Universal Robots PolyScope program: PaintTop.urp

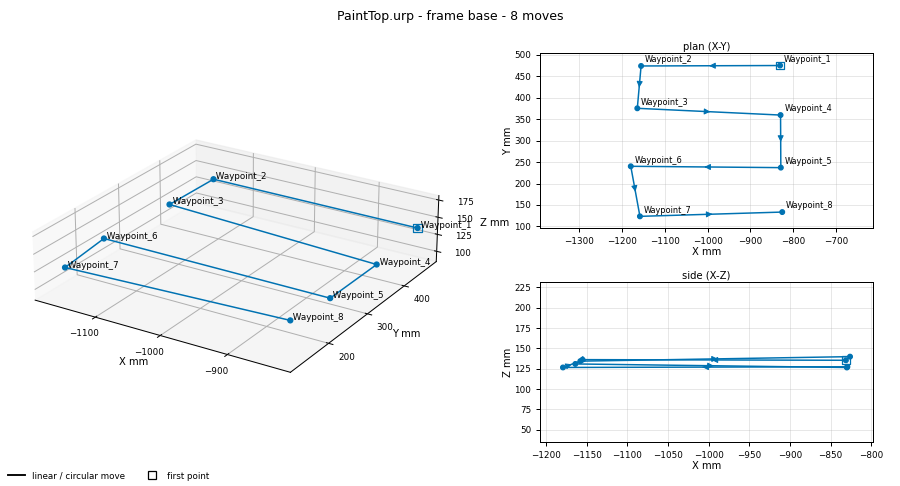
[picture p0: tool path of PaintTop.urp in frame base, 8 of 8 moves have a stored position in this frame; points joined in program order, loops and branches not executed]
Program PaintTop (createdIn=3.0.0 lastSavedIn=3.0.0 directory=/programs installation=default)
Robot Program (runOnlyOnce=true motionType=MoveJ speed=1.047198 acceleration=1.396263 useActiveTCP=false)
  'Program generated by RoboDK v5.6.4 for UR10 on 06/12/2023 15:16:24'
  'Using nominal kinematics.'
  'Using Ref. Frame 2: p[-0.800000, 0.500000, 0.100000, 0.000000, 0.000000, 3.141593]'
  'Using TCP Paint gun: p[0.050000, 0.000000, 0.450000, 0.000000, 0.523599, 0.000000]'
  Script: set_tcp(p[0.050000, 0.000000, 0.450000, 0.000000, 0.523599, 0.000000])
  Script: movej([-3.831626, -2.007006, -1.342958, -1.224118, 2.230775, 1.418370],1.20000,0.75000,0,0.0000)
  MoveJ speed 42.97 deg/s, acceleration 68.75 deg/s^2 (useActiveTCP=true)
    Waypoint Waypoint_1: TCP in base x=-831.072 y=475.215 z=135.355 mm, rx=2.4575 ry=-0.3994 rz=0.1361 rad; joints [-219.536, -114.993, -76.946, -70.137, 127.814, 81.267] deg; flange x=-658.722 y=682.921 z=498.885 mm, rx=2.4703 ry=-0.6178 rz=-0.5174 rad
  MoveL speed 50 mm/s, acceleration 1200 mm/s^2 (useActiveTCP=true)
    Waypoint Waypoint_2: TCP in base x=-1155.2 y=474.185 z=136.15 mm, rx=2.4708 ry=-0.2859 rz=0.0974 rad; joints [-210.289, -143.985, -30.818, -80.427, 128.618, 88.068] deg; flange x=-978.302 y=694.591 z=489.884 mm, rx=2.4592 ry=-0.5038 rz=-0.5561 rad
    Waypoint Waypoint_3: TCP in base x=-1164.047 y=375.424 z=130.832 mm, rx=-2.7996 ry=0.4397 rz=0.0688 rad; joints [-179.629, -118.486, -75.308, -44.885, 65.562, 96.641] deg; flange x=-991.095 y=195.639 z=508.674 mm, rx=-2.636 ry=0.3054 rz=0.7762 rad
    Waypoint Waypoint_4: TCP in base x=-829.883 y=359.668 z=126.469 mm, rx=-2.8183 ry=0.5893 rz=0.0791 rad; joints [-177.894, -88.354, -112.979, -39.189, 64.009, 104.945] deg; flange x=-663.406 y=180.05 z=507.287 mm, rx=-2.6304 ry=0.4588 rz=0.7846 rad
    Waypoint Waypoint_5: TCP in base x=-829.25 y=237.038 z=127.37 mm, rx=2.8595 ry=-0.3065 rz=0.0412 rad; joints [-194.064, -91.552, -105.349, -45.917, 103.957, 95.559] deg; flange x=-651.679 y=309.287 z=537.551 mm, rx=2.8239 ry=-0.4027 rz=-0.7133 rad
    Waypoint Waypoint_6: TCP in base x=-1179.268 y=240.16 z=126.516 mm, rx=2.8673 ry=-0.2142 rz=0.0288 rad; joints [-190.188, -122.622, -65.046, -54.105, 103.992, 95.944] deg; flange x=-999.586 y=323.516 z=533.66 mm, rx=2.8148 ry=-0.3107 rz=-0.724 rad
    Waypoint Waypoint_7: TCP in base x=-1157.907 y=123.396 z=134.284 mm, rx=-2.4798 ry=0.1696 rz=0.0578 rad; joints [-157.813, -118.488, -80.898, -50.291, 43.391, 100.711] deg; flange x=-977.901 y=-149.455 z=447.573 mm, rx=-2.3736 ry=-0.0548 rz=0.6957 rad
    Waypoint Waypoint_8: TCP in base x=-825.987 y=133.387 z=139.825 mm, rx=-2.6833 ry=0.2664 rz=0.0605 rad; joints [-153.215, -84.837, -115.212, -52.717, 50.654, 115.012] deg; flange x=-647.834 y=-77.956 z=498.427 mm, rx=-2.5528 ry=0.0987 rz=0.7461 rad
